FUNCTION FC_Check_IN : BOOL
VAR_INPUT
	I_sString : REFERENCE TO T_MaxString;
END_VAR
VAR
	stringPos	: INT;
END_VAR

stringPos := FIND(I_sString, 'IN');
IF stringPos <> 0 THEN
	I_sString := MID(I_sString, LEN(I_sString), stringPos+1);
	FC_Check_IN := TRUE;
ELSE
	FC_Check_IN := FALSE;
END_IF

END_FUNCTION

(* stored: Version 1.1.0.1, ProductVersion 3.1.4024.15
   POU FC_Check_IN: Id {e19346fb-ee03-4b8b-8067-be87365ee801}, SpecialFunc None *)
